FUNCTION_BLOCK FB_TcpIpComm EXTENDS T_NamedBase IMPLEMENTS I_BootService
VAR_INPUT
END_VAR
VAR_OUTPUT
END_VAR
VAR
  // boot service
  _bStarting       : BOOL := TRUE;
  _tStartDelay     : ARRAY[1..nMaxTcpIpClients] OF TIME;
  fbTonStartDelay  : ARRAY[1..nMaxTcpIpClients] OF TON;
  
  // TcpIp clients list
  sSrvNetId        : T_AmsNetID := '';           (* AmsId of tcpip server.exe, default: empty string. *)
  fbCloseAll       : FB_SocketCloseAll;          (* close all opened sockets *)
  
  fbTcpClients     : ARRAY[1..nMaxTcpIpClients] OF FB_TcpClient;
  pActiveClients   : ARRAY[1..nMaxTcpIpClients] OF POINTER TO FB_TcpClient;
  nActiveTcpClients: UINT;    // active/registered clients¨
  
  nCtr  : UINT;
END_VAR
VAR CONSTANT
  nMaxTcpIpClients      : UINT := 4;
END_VAR

IF _bStarting THEN RETURN; END_IF

// call all active clients
FOR nCtr:=1 TO nActiveTcpClients DO
  fbTonStartDelay[nCtr](IN := TRUE, PT := _tStartDelay[nCtr]);
  IF fbTonStartDelay[nCtr].Q THEN
    fbTcpClients[nCtr](
      //bEnable := .....
      //bConnected => 
    );
  END_IF
END_FOR

PROPERTY bStarting : BOOL
GET
// return booint satus to boot service
bStarting := _bStarting;
END_GET
END_PROPERTY

METHOD closeAllSockets : BOOL
VAR_INST
  bClosing  : BOOL;
END_VAR
(* close all opened/created sockets *)
IF NOT bClosing THEN fbCloseAll( sSrvNetId := sSrvNetId, bExecute:= FALSE ); bClosing := TRUE; END_IF  // be sure to call it once with FALSE

fbCloseAll( sSrvNetId := sSrvNetId, bExecute:= bClosing );
IF NOT fbCloseAll.bBusy THEN
  // done
  //IF fbCloseAll.bError THEN LogError(F_Concat2('CloseAllSockets error=', F_GetAdsErrDescription(lErrCode:=fbCloseAll.nErrId))); 
  //ELSE                      LogInfo('CloseAllSockets done.'); END_IF
  bClosing := FALSE;
END_IF

// return busy
closeAllSockets := fbCloseAll.bBusy;
END_METHOD

METHOD registerTcpIpClient : POINTER TO FB_TcpClient
VAR_INPUT
  sRemoteHost   : ST_SockAddr;
  iHandler      : I_TcpIp_RxMsgHandler;
  tStartDelay   : TIME;
END_VAR

VAR
  pTcpIpClient  : POINTER TO FB_TcpClient;
END_VAR
IF nActiveTcpClients >= nMaxTcpIpClients THEN
  LogError('No free TcpIp client, ignore registerTcpIpClient');
END_IF

nActiveTcpClients := nActiveTcpClients + 1;

// config
fbTcpClients[nActiveTcpClients].sRemoteHost := sRemoteHost.sAddr;
fbTcpClients[nActiveTcpClients].nRemotePort := sRemoteHost.nPort;
_tStartDelay[nActiveTcpClients]             := tStartDelay;

// init
fbTcpClients[nActiveTcpClients].init(
  tReconnect := T#100MS,
  tRxPolling := T#1MS,
  //cMsgTermination := cMSG_TERMINATION_ZERO
);
// start
fbTcpClients[nActiveTcpClients].bEnable := TRUE;
fbTcpClients[nActiveTcpClients].register_RxMsgHandler(bAdd:=TRUE, iHandler);

// return client handle (pointer = full access)
pActiveClients[nActiveTcpClients] := ADR(fbTcpClients[nActiveTcpClients]);
registerTcpIpClient := ADR(fbTcpClients[nActiveTcpClients]);
END_METHOD

METHOD start : BOOL
// called by system boot services, 'regBootService' needed
IF NOT closeAllSockets() THEN
  // done 
  _bStarting := FALSE;  // we are done
END_IF

start := _bStarting;
END_METHOD

END_FUNCTION_BLOCK

(* stored: Version 1.1.0.1, ProductVersion 3.1.4024.3
   POU FB_TcpIpComm: Id {a078388e-b697-4203-9214-41bca8598ae3}, SpecialFunc None
   Folder I_BootService: Id {8dae093d-9041-4467-8abd-4c2547d9939f}
   Property bStarting: Id {75b53b4f-1b56-40c9-84b6-ac5f91952b36}
   Get Get: Id {aad467fa-61af-4801-bffc-b0fc09a43449}
   Method closeAllSockets: Id {44728c69-93f7-4a0a-b50f-7543336635d2}
   Method registerTcpIpClient: Id {615b5775-a0f2-4292-abc2-3bb5e0b363cd}
   Method start: Id {20fbdb4a-e6fc-4b98-8d94-a8b0f07207dc} *)
